PROGRAM MAIN
VAR
	// Here, the detector, reject arm, and memory for detection are created as BOOLs
	bBadPartDetected: BOOL := FALSE;
	bRejectArmEnabled: BOOL := FALSE;
	bRejectMemory: BOOL := FALSE;
	
	// Timers to calculate when to enable the reject arm are made here.
	tTravelTimer: TON;
	tPushTimer: TON;
	
END_VAR

//Detects if a faulty product is detected and saves a memory variable for it.
IF bBadPartDetected THEN
	bRejectMemory := TRUE;
END_IF;

// Timer is then enabled while setting an if statement to enable/disable the reject arm.
tTravelTimer(IN:= bRejectMemory, PT := T#3S);
tPushTimer(IN:= tTravelTimer.Q, PT:= T#1S);

IF NOT tPushTimer.Q AND bRejectMemory AND tTravelTimer.Q THEN
	bRejectArmEnabled := TRUE;
ELSE;
	bRejectArmEnabled := FALSE;
END_IF;

//When all timers are completed, both start conditions are set to false, reseting the cycle.
IF tPushTimer.Q AND tTravelTimer.Q THEN
	bBadPartDetected := FALSE;
	bRejectMemory := FALSE;
END_IF;

END_PROGRAM

(* stored: Version 1.1.0.1, ProductVersion 3.1.4024.16
   POU MAIN: Id {83d9dde9-3524-4855-af7f-721d30e69b7f}, SpecialFunc None *)
